# EPICS substitutions: ipmiMgrApp/Db/rtm_8sfp.substitutions
#
# RTM 8SFP
#

#nat> show_sensorinfo 90
#Sensor Information for FRU 90 / RTM1
#==================================================================
#  #   SDRType  Sensor Entity Inst  Value   State    Name
#------------------------------------------------------------------
#  -   MDevLoc          0xc0  0x67                    AFC Timing-RTM
# 20   Compact  0xf2    0xc0  0x67  0xa1              HOTSWAP RTM
# 21   Full     Temp    0xc0  0x67  30.0 C     ok     TEMP RTM1
# 22   Full     Temp    0xc0  0x67  29.5 C     ok     TEMP RTM2
# 23   Compact  0xf0    0xc0  0x61  0x02              HS 090 RTM1
# ------------------------------------------------------------------

file "fru_common_alias.db"
{
   pattern { id    , fruid    }
           { $(id) , $(fruid) }
}

file "sensor_ai_alias.db"
{
    pattern { attr        , sensinst , type , fruid    , prefix  , aliasprefix  }
            { TempRTM1    , 1        , 1    , $(fruid) , $(id)   , alias_$(id)        }
            { TempRTM2    , 2        , 1    , $(fruid) , $(id)   , alias_$(id)        }
}
